// TwinCAT 3 PLC project PRG_Test_Periphery
// Company: RafalOS
// ProgramVersion: 3.1.4024.0
// libraries:
//   B_Actuator, * (RafalOS)
//   B_Base, * (RafalOS)
//   B_IO, * (RafalOS)
//   B_IODecorator, * (RafalOS)
//   Tc2_DataExchange, * (Beckhoff Automation GmbH)
//   Tc2_Standard, * (Beckhoff Automation GmbH)
//   Tc2_System, * (Beckhoff Automation GmbH)
//   Tc3_Module, * (Beckhoff Automation GmbH)
//   TcUnit, * (www.tcunit.org)
// project tree:
//   GVLs/ GVL_Actuator.TcGVL (not stored), GVL_Decorators.TcGVL, GVL_Variable.TcGVL
//   / PlcTask.TcTTO (not stored)
//   POUs/ FB_ActuatorTest.TcPOU (not stored), FB_ButtonTest.TcPOU (not stored), FB_ElectroValveTest.TcPOU (not stored), FB_LampBlinkingTest.TcPOU (not stored), FB_SensorDecoratorTestTest.TcPOU, FB_SensorTest.TcPOU (not stored)
//   TESTs/ PRG_Test.TcPOU
// real-time tasks:
//   TASK PlcTask: cycle T#10ms, priority 20, ADS port 350

// ---- GVLs/GVL_Decorators.TcGVL
{attribute 'qualified_only'}
VAR_GLOBAL
	senNO				: FB_Sensor_NO;
	senNC				: FB_Sensor_NC;
	senNO_2inRow		: FB_Sensor_NO_2InRow;
	
	senNO_TestDecorator			: FB_Sensor_NO_TestDecorator (fbToDecorate := senNO);
	senNC_TestDecorator			: FB_Sensor_NC_TestDecorator (fbToDecorate := senNC);
	senNO_2inRow_TestDecorator	: FB_Sensor_NO_2InRow_TestDecorator (fbToDecorate := senNO_2inRow);
	
END_VAR

// ---- GVLs/GVL_Variable.TcGVL
{attribute 'qualified_only'}
VAR_GLOBAL
	fbSaveDataByADS		: Tc2_DataExchange.FB_WriteAdsSymByName;
	bValueToSave		: BOOL;
	bSaved				: BOOL;
	bSave				: BOOL;
	sData				: STRING;
//Czujników	
	senNC				: FB_Sensor_NC;
	senNO				: FB_Sensor_NO;
	sen2NO				: FB_Sensor_NO_2InRow;
//TEST Elektrozawor
	ev3on2_NC			: FB_Electrovalve_3on2_NC;
	ev3on2_NO			: FB_Electrovalve_3on2_NO;
	ev5on2_1C			: FB_Electrovalve_5on2_1Coil;
	ev5on2_2C			: FB_Electrovalve_5on2_2Coil;
	ev5on3_2C_ven		: FB_Electrovalve_5on3_2Coil_Vented;
	ev5on3_2C_inf		: FB_Electrovalve_5on3_2Coil_Infected;
//
	fbLampBlinking		: FB_LampBlinking;
//
	fbButton_NC				: FB_Button_NC;
	fbButton_NO				: FB_Button_NO;

END_VAR

// ---- POUs/FB_SensorDecoratorTestTest.TcPOU
FUNCTION_BLOCK FB_SensorDecoratorTestTest EXTENDS TcUnit.FB_TestSuite
VAR

END_VAR


T01_TestCzujnikNC ();
T02_TestCzujnikNO ();
T03_TestCzujnikNO_Szereg ();

METHOD PROTECTED T01_TestCzujnikNC
VAR_INST
	iKrok		: INT;
END_VAR
IF (TcUnit.TEST_ORDERED ('T01_TestCzujnikNC')) THEN
	GVL_Decorators.senNC_TestDecorator.SetContact (bIN := TRUE);
	AssertFalse (Condition := GVL_Decorators.senNC_TestDecorator.IsActive (), Message := 'T11 - bledny stan');
	GVL_Decorators.senNC_TestDecorator.SetContact (bIN := FALSE);
	AssertTrue (Condition := GVL_Decorators.senNC_TestDecorator.IsActive (), Message := 'T12 - bledny stan');
	GVL_Decorators.senNC_TestDecorator.SetContact (bIN := TRUE);
	AssertFalse (Condition := GVL_Decorators.senNC_TestDecorator.IsActive (), Message := 'T13 - bledny stan');
	
	TcUnit.TEST_FINISHED ();
END_IF
END_METHOD

METHOD PROTECTED T02_TestCzujnikNO
VAR_INST
	iKrok		: INT;
END_VAR
IF (TcUnit.TEST_ORDERED ('T02_TestCzujnikNO')) THEN
	GVL_Decorators.senNO_TestDecorator.SetContact (bIN := FALSE);
	AssertFalse (Condition := GVL_Decorators.senNo_TestDecorator.IsActive (), Message := 'T11 - bledny stan');
	GVL_Decorators.senNO_TestDecorator.SetContact (bIN := TRUE);
	AssertTrue (Condition := GVL_Decorators.senNO_TestDecorator.IsActive (), Message := 'T12 - bledny stan');
	GVL_Decorators.senNO_TestDecorator.SetContact (bIN := FALSE);
	AssertFalse (Condition := GVL_Decorators.senNO_TestDecorator.IsActive (), Message := 'T13 - bledny stan');

	TcUnit.TEST_FINISHED ();
END_IF
END_METHOD

METHOD PROTECTED T03_TestCzujnikNO_Szereg
VAR_INST
	ikrok			: int;
END_VAR
IF (TcUnit.TEST_ORDERED ('T03_TestCzujnikNO_Szereg')) THEN
	GVL_Decorators.senNO_2inRow_TestDecorator.SetContact (bIN := FALSE);
	GVL_Decorators.senNO_2inRow_TestDecorator.SetContact2 (bIN := FALSE);
	AssertFalse (Condition := GVL_Decorators.senNO_2inRow_TestDecorator.IsActive (), Message := 'T11 - bledny stan');
	
	GVL_Decorators.senNO_2inRow_TestDecorator.SetContact (bIN := TRUE);
	AssertFalse (Condition := GVL_Decorators.senNO_2inRow_TestDecorator.IsActive (), Message := 'T12 - bledny stan');

	GVL_Decorators.senNO_2inRow_TestDecorator.SetContact2 (bIN := TRUE);
	AssertTrue (Condition := GVL_Decorators.senNO_2inRow_TestDecorator.IsActive (), Message := 'T13 - bledny stan');

	GVL_Decorators.senNO_2inRow_TestDecorator.SetContact (bIN := FALSE);
	AssertFalse (Condition := GVL_Decorators.senNO_2inRow_TestDecorator.IsActive (), Message := 'T14 - bledny stan');

	GVL_Decorators.senNO_2inRow_TestDecorator.SetContact2 (bIN := FALSE);
	AssertFalse (Condition := GVL_Decorators.senNO_2inRow_TestDecorator.IsActive (), Message := 'T15 - bledny stan');
	
	TcUnit.TEST_FINISHED ();
END_IF
END_METHOD

END_FUNCTION_BLOCK

// ---- TESTs/PRG_Test.TcPOU
PROGRAM PRG_Test
VAR
	fbSensorTest			: FB_SensorTest;
	fbElectrovalveTest		: FB_ElectroValveTest;
	fbButtontest			: FB_ButtonTest;
	fbLapmBlinkingTest		: FB_LampBlinkingTest;
	
	fbActuatortest			: FB_ActuatorTest;
	
	fbSensortestDecoratorTest	: FB_SensorDecoratorTestTest;
	
END_VAR


	TcUnit.RUN_IN_SEQUENCE ();


GVL_Variable.fbSaveDataByADS (
	bWrite		:= GVL_Variable.bSave,
	sNetId		:= ,
	nPort		:= ,
	sVarName	:= GVL_Variable.sData,
	nSrcAddr	:= ADR (GVL_Variable.bValueToSave),
	nLen		:= SIZEOF (GVL_Variable.bValueToSave),
	tTimeout	:= ,
	eComMode	:= ,
	bBusy		=> GVL_Variable.bSaved,
	bError		=> ,
	nErrorId	=>
);

END_PROGRAM
